// TIA Portal V18 export
VAR_GLOBAL   // PLC tag table "04_10 Costanti Nomi Attuatore Stz10"
END_VAR
VAR_GLOBAL CONSTANT   // user constants
   P1001 : Int := 1;   // EV salita discesa scarico 1
   P1002 : Int := 2;   // EV salita discesa scarico 2
   P1003 : Int := 3;   // EV salita discesa scarico 3
   EVSCARICO1 : Int := 4;   // EV scarico 1
   EVSCARICO2 : Int := 5;   // EV scarico 2
   EVSCARICO3 : Int := 6;   // EV scarico 3
   EVSCARICO4 : Int := 7;   // EV scarico 4
END_VAR
